// TwinCAT 3 PLC project Untitled1
// ProgramVersion: 3.1.4023.0
// libraries:
//   Tc2_Standard, * (Beckhoff Automation GmbH)
//   Tc2_System, * (Beckhoff Automation GmbH)
//   Tc2_Utilities, * (Beckhoff Automation GmbH)
//   Tc3_Module, * (Beckhoff Automation GmbH)
// project tree:
//   DUTs/ HMI_Button.TcDUT, HMI_Instructions.TcDUT, IO_Struct.TcDUT, Port_Map.TcDUT, SL_INSTRUCTIONS.TcDUT, Test_Log.TcDUT
//   GVLs/ GVL_HMI.TcGVL, GVL_IO_STRUCTS.TcGVL, GVL_LOGS.TcGVL, GVL_IO.TcGVL, CONSTANTS.TcGVL
//   / PlcTask.TcTTO
//   POUs/ FB_EXECUTE_SECTION1.TcPOU, FB_EXECUTE_SECTION2.TcPOU, INITIALIZE.TcPOU, LOG_SECTION2.TcPOU, LOG_SECTION1.TcPOU, MAIN.TcPOU, UNINITIALIZE.TcPOU, WRITE_IO_VALUES.TcPOU
// real-time tasks:
//   TASK PlcTask: cycle T#10ms, priority 20, ADS port 350
// I/O:
//   DEVICE Device 1 (EtherCAT), AmsNetId 169.254.202.152.2.1
//     C0 (EK1914) [EK1914, 2 Ch. Safety Input/Output 24V,  TwinSAFE]
//       modules: Module 1 (FSOE), Module 2 (DIO)
//       C1 (EL9410) [EL9410 E-Bus Power Supplier  (Diagnostics)]
//       C2 (EL2014) [EL2014 4Ch. Dig. Output 24V, 0,5A, Diagnostic]
//       C3 (EL1018) [EL1018 8Ch. Dig. Input 24V, 10µs]
//       C4 (EL1819) [EL1819 16Ch. Dig. Input 24V, 10µs]
//       C5 (EL1819) [EL1819 16Ch. Dig. Input 24V, 10µs]
//       C6 (EK1122-0008) [EK1122-0008 2 port EtherCAT junction M8]
//         JBC0 (EK1914) [EK1914, 2 Ch. Safety Input/Output 24V,  TwinSAFE]
//           modules: Module 1 (FSOE), Module 2 (DIO)
//           JBC1 (EL9410) [EL9410 E-Bus Power Supplier  (Diagnostics)]
//           JBC2 (EL1904) [EL1904, 4 Ch. Safety Input 24V, TwinSAFE]
//             modules: Module 1 (FSOES)
//           JBC3 (EL3174) [EL3174 4K. Ana. Eingang  +/-10V Diff., +/-20mA SingleEnded, 16 Bit]
//           JBC4 (EK1122-0008) [EK1122-0008 2 port EtherCAT junction M8]
//           JBC5 (EK1122-0008) [EK1122-0008 2 port EtherCAT junction M8]
//             Box 14 (EP3752-0000) [EP3752-0000 Acceleration Sensor]
// variable links:
//   Untitled1/Untitled1 Instance <-> Device 1 (EtherCAT)/C0 (EK1914)/C2 (EL2014)
//     PlcTask Outputs/GVL_IO.SF5_Fire_Alarm <-> DIG Outputs/Channel 2/Output
//   Untitled1/Untitled1 Instance <-> Device 1 (EtherCAT)/C0 (EK1914)/C3 (EL1018)
//     PlcTask Inputs/GVL_IO.J7_24V_Up <-> Channel 1/Input
//     PlcTask Inputs/GVL_IO.J8_24V_Up <-> Channel 3/Input
//     PlcTask Inputs/GVL_IO.J7_24V_Us <-> Channel 6/Input
//     PlcTask Inputs/GVL_IO.J8_24V_Us <-> Channel 8/Input
//   Untitled1/Untitled1 Instance <-> Device 1 (EtherCAT)/C0 (EK1914)/C4 (EL1819)
//     PlcTask Inputs/GVL_IO.J{1..6}_24V_Up <-> Channel {1..11 step 2}/Input  (6 links)
//     PlcTask Inputs/GVL_IO.J{1..6}_24V_Us <-> Channel {2..12 step 2}/Input  (6 links)
//   Untitled1/Untitled1 Instance <-> Device 1 (EtherCAT)/C0 (EK1914)/C5 (EL1819)
//     PlcTask Inputs/GVL_IO.SF1_MF_CONTINUITY <-> Channel 16/Input
//     PlcTask Inputs/GVL_IO.SF2_MF_CONTINUITY <-> Channel 15/Input
//     PlcTask Inputs/GVL_IO.SF4_Pull_Station <-> Channel 14/Input
//     PlcTask Inputs/GVL_IO.SF6_MGT_CONTINUITY <-> Channel 13/Input
//     PlcTask Inputs/GVL_IO.SF8_MGT_CONTINUITY <-> Channel 12/Input
//   Untitled1/Untitled1 Instance <-> Device 1 (EtherCAT)/C0 (EK1914)/C6 (EK1122-0008)/JBC0 (EK1914)
//     PlcTask Inputs/GVL_IO.JB_DCDCS_OK <-> Module 2 (DIO)/DIO Inputs/Input 0
//     PlcTask Inputs/GVL_IO.JB_Door_Switch <-> Module 2 (DIO)/DIO Inputs/Input 1
//     PlcTask Inputs/GVL_IO.JB_PSU1_OK <-> Module 2 (DIO)/DIO Inputs/Input 2
//     PlcTask Inputs/GVL_IO.JB_PSU2_OK <-> Module 2 (DIO)/DIO Inputs/Input 3

CONFIGURATION Untitled1
    RESOURCE PLC ON TwinCAT3
        TASK PlcTask(INTERVAL := T#10ms, PRIORITY := 20);
        PROGRAM MAIN WITH PlcTask : MAIN;
    END_RESOURCE
END_CONFIGURATION

// ---- DUTs/HMI_Button.TcDUT
TYPE HMI_Button :
STRUCT
	Text : STRING(50);
	Live_Value : BOOL;
END_STRUCT
END_TYPE

// ---- DUTs/HMI_Instructions.TcDUT
TYPE HMI_Instructions :
STRUCT
	Instructions : STRING(200);
	Status : BOOL;
END_STRUCT
END_TYPE

// ---- DUTs/IO_Struct.TcDUT
TYPE IO_Struct :
STRUCT
	SECTION : INT;
	INDEX : INT;
	CARD : STRING(10);
	TERMINAL : USINT;
	SCH_LBL : STRING(10);
	Signal : STRING(25);
	TESTER_PORT : STRING(10);
	TARGET_PORT : STRING(10);
	DESCRIPTION : STRING(255);
	LIVE_BOOL : BOOL;
	LIVE_INT : INT;
	EXPECTED_BOOL : BOOL;
	EXPECTED_INT : INT;
	RESULT : STRING(10);
END_STRUCT
END_TYPE

// ---- DUTs/Port_Map.TcDUT
TYPE Port_Map :
STRUCT
	JBOX_PORT : STRING(5);
	TESTER_PORT : STRING(5);
END_STRUCT
END_TYPE

// ---- DUTs/SL_INSTRUCTIONS.TcDUT
TYPE SL_INSTRUCTIONS :
STRUCT
	Line : STRING(255);
END_STRUCT
END_TYPE

// ---- DUTs/Test_Log.TcDUT
TYPE Test_Log :
STRUCT
	Index : INT;
	Description : STRING(255);
	Result : STRING(10);
END_STRUCT
END_TYPE

// ---- GVLs/GVL_HMI.TcGVL
{attribute 'qualified_only'}
VAR_GLOBAL
	
	JBOX_TEST_PORT_MAP : ARRAY[0..CONSTANTS.NUM_CONNECTIONS-1] OF Port_Map := [
		(
			JBOX_PORT := 'J37',
			TESTER_PORT := 'SF1'
		),
		(
			JBOX_PORT := 'S2',
			TESTER_PORT := 'SF2'
		),
		(
			JBOX_PORT := 'S33',
			TESTER_PORT := 'J1'
		),
		(
			JBOX_PORT := 'S34',
			TESTER_PORT := 'J2'
		),
		(
			JBOX_PORT := 'S25',
			TESTER_PORT := 'J3'
		),
		(
			JBOX_PORT := 'S26',
			TESTER_PORT := 'J4'
		),
		(
			JBOX_PORT := 'S27',
			TESTER_PORT := 'J5'
		),
		(
			JBOX_PORT := 'S28',
			TESTER_PORT := 'J6'
		),
		(
			JBOX_PORT := 'S29',
			TESTER_PORT := 'J7'
		),
		(
			JBOX_PORT := 'S30',
			TESTER_PORT := 'J8'
		),
		(
			JBOX_PORT := 'S1',
			TESTER_PORT := 'J9'
		),
		(*
		(
			JBOX_PORT := 'S35',
			TESTER_PORT := 'J10'
		),
		*)
		(
			JBOX_PORT := 'S3',
			TESTER_PORT := 'J11'
		),
		(
			JBOX_PORT := 'S5',
			TESTER_PORT := 'J12'
		),
		(
			JBOX_PORT := 'S8',
			TESTER_PORT := 'J13'
		),
		(
			JBOX_PORT := 'S10',
			TESTER_PORT := 'J14'
		),
		(
			JBOX_PORT := 'S21',
			TESTER_PORT := 'J15'
		),
		(
			JBOX_PORT := 'S22',
			TESTER_PORT := 'J16'
		),
		(
			JBOX_PORT := 'S23',
			TESTER_PORT := 'J17'
		),
		(
			JBOX_PORT := 'S24',
			TESTER_PORT := 'J18'
		),
		(
			JBOX_PORT := 'S4',
			TESTER_PORT := 'J19'
		),
		(
			JBOX_PORT := 'S6',
			TESTER_PORT := 'J20'
		),
		(
			JBOX_PORT := 'S9',
			TESTER_PORT := 'J21'
		),
		(
			JBOX_PORT := 'S11',
			TESTER_PORT := 'J22'
		),
		(
			JBOX_PORT := 'S13',
			TESTER_PORT := 'J23'
		),
		(
			JBOX_PORT := 'S14',
			TESTER_PORT := 'J24'
		),
		(
			JBOX_PORT := 'S15',
			TESTER_PORT := 'J25'
		),
		(
			JBOX_PORT := 'S16',
			TESTER_PORT := 'J26'
		),
		(
			JBOX_PORT := 'J36',
			TESTER_PORT := 'S17'
		)
		(*
		(
			JBOX_PORT := 'J38',
			TESTER_PORT := 'S18'
		)
		*)
		];

	//
	//
	//
	
	(*
	HMI_HOME_INSTRUCTIONS : ARRAY[0..1] OF HMI_INSTRUCTIONS := [
	];
	*)
	
	HMI_HOME_INSTRUCTIONS : ARRAY[0..CONSTANTS.HMI_HOME_NUM_INSTRUCTIONS-1] OF HMI_INSTRUCTIONS := [
		(Instructions := 'Place JBOX Next to Acceptance Tester',
		 Status := FALSE),
		(Instructions := 'Visually inspect the box for foreign objects, floating wires, or any signs of being incomplete',
		 Status := FALSE),
		(Instructions := 'Unplug power from the acceptance tester',
		 Status := FALSE),
		(Instructions := 'Verify green bonding wire is present to bond the door to the enclosure',
		 Status := FALSE),
		(Instructions := 'Connect All Tester Cables to JBOX Ports as Shown in the Port Map, Leave 120V Disconnected',
		 Status := FALSE),
		(Instructions := 'Open All Breakers in Acceptance Tester Panel',
		 Status := FALSE),
		(Instructions := 'Supply 480V Weld Plug on Acceptance Tester with 480V Power',
		 Status := FALSE),
		(Instructions := 'Close All Breakers in Acceptance Tester Panel',
		 Status := FALSE)
		 
	];
	
	HMI_HOME_BEGIN_TEST_BUTTON : HMI_BUTTON := (
		Text := 'Initiate JBOX Test',
		Live_Value := FALSE
	);
	
	HMI_SECTION_1_INSTRUCTIONS : ARRAY[0..CONSTANTS.HMI_SECTION_1_NUM_INSTRUCTIONS-1] OF HMI_INSTRUCTIONS := [
		(Instructions := 'Verify 480V Indicator for JBOX on Acceptance Tester',
		 Status := FALSE),
		(Instructions := 'Perform PSU1 Configuration',
		 Status := FALSE),
		(Instructions := 'Perform DCDC1 Configuration',
		 Status := FALSE),
		(Instructions := 'Perform DCDC2 Configuration',
		 Status := FALSE),
		(Instructions := 'Open JBOX Door',
		 Status := FALSE),
		(Instructions := 'Press Estop',
		 Status := FALSE),
		(Instructions := 'Pull Fire Alarm',
		 Status := FALSE)
	];
	
	HMI_PSU_CONFIG_INSTRUCTIONS : ARRAY[0..13] OF SL_INSTRUCTIONS := [
		(Line := 'Open the Phoenix Contact "Quint Power" App'),
		(Line := 'Install temportary 22 AWG jumper wire from PSU2 Rem signal to 0V TB'),
		(Line := 'Select READ VIA NFC'),
		(Line := 'Select SCAN VIA NFC'),
		(Line := 'Place top edge of phone over the QR code on PSU2 until power supply is read successfully'),
		(Line := 'Select OUTPUT VOLTAGE menu'),
		(Line := 'Set OUTPUT VOLTAGE to 26.00V'),
		(Line := 'Set PARALLEL OPERATION to TRUE'),
		(Line := 'Exit OUTPUT VOLTAGE menu and select SIGNALING menu'),
		(Line := 'Set OUT 2 to ANALOG OUTPUT with OUTPUT CURRENT'),
		(Line := 'Exit SIGNALING menu'),
		(Line := 'Select NFC button and plade top edge of phone over the QR code on PSU1 until the dara is written succesfully'),
		(Line := 'Remove temportary 22 AWG jumper wire FROM PSU2 Rem signal TO 0V TB'),
		(Line := 'Close Quint Power App')
	];
	
	HMI_DCDC_CONFIG_INSTRUCTIONS : ARRAY[0..3] OF SL_INSTRUCTIONS := [
		(Line := 'Pull ferrules inserted into terminals 2.1 and 2.2 in DC/DC slightly out so you can probe voltage on exposed ferrule'),
		(Line := 'Turn Uout dial on DC/DC2 until the DC/DCs output is 52V. Probe on exposed ferrules to verify'),
		(Line := 'Reseat ferrules to correct depth'),
		(Line := 'Write "52V, todays DATE, your initials" on the label on DC/DC')
	];

	
	
	HMI_SECTION_1_BEGIN_AUTOMATED_BUTTON : HMI_BUTTON := (
		Text := 'Begin Automated Test',
		Live_Value := FALSE
	);
	
	HMI_SECTION_2_INSTRUCTIONS : ARRAY[0..CONSTANTS.HMI_SECTION_2_NUM_INSTRUCTIONS-1] OF HMI_INSTRUCTIONS := [
		(Instructions := 'Reset Estop',
		 Status := FALSE),
		(Instructions := 'Reset Fire Alarm, use the key tied to the top of the acceptance tester to open the box and reset it',
		 Status := FALSE),
		(Instructions := 'Unplug J36 and S1 Connections on JBOX',
		 Status := FALSE),
		(Instructions := 'Plug J10 and S18 From Acceptance Tester into JBOX S35 and J38 Respectively',
		 Status := FALSE),
		(Instructions := 'Perform PSU2 Configuration',
		 Status := FALSE),
		(Instructions := 'Verify 120V Indicator for JBOX on Acceptance Tester',
		 Status := FALSE),
		(Instructions := 'Verify 120V Indicator FOR GRACE Port Verification Lit Up',
		 Status := FALSE),
		 (Instructions := 'Close JBOX Door',
		 Status := FALSE)
	];
	
	HMI_SECTION_2_BEGIN_AUTOMATED_BUTTON : HMI_BUTTON := (
		Text := 'Begin Automated Test',
		Live_Value := FALSE
	);
	
	
	HMI_ABORT_TEST_BUTTON : HMI_BUTTON := (
		Text := 'ABORT JBOX TEST',
		Live_Value := FALSE
	);
	
	HMI_RESET_TEST_BUTTON : HMI_BUTTON := (
		Text := 'Reset Jbox Test',
		Live_Value := FALSE
	);
	

	ACTIVE_HMI_VIEW_STRING : STRING(50);
	
	ACTIVE_HMI_VIEW : INT := 0;

	
	



	
	
END_VAR

// ---- GVLs/GVL_IO_STRUCTS.TcGVL
{attribute 'qualified_only'}
VAR_GLOBAL
	
	
	// STILL NEED ESTOP VERIFICATION, PSU VERIFICATION, DCDC VERIFICATION

	// SECTION ONE OCCURS WITH DOOR CLOSED AND ESTOP DEPRESSED AND NOTHING CONFIGURED
	IO_MAP_SECTION1_DIG : ARRAY[0..CONSTANTS.SECTION1_NUM_DIG_TESTS-1] OF IO_STRUCT := [
		(
			SECTION := 1,
			INDEX := 0,
			SCH_LBL := 'J7_4',
			SIGNAL := 'Digital',
			TESTER_PORT := 'J7',
			DESCRIPTION := '480V Supplied 7/8 S29 Up 24V Power Check', // This is written to HMI
			LIVE_BOOL := 0, // This is written to from the IO variable
			EXPECTED_BOOL := 1,
			RESULT := 'FAIL' // This is written from HMI
		),
		(
			SECTION := 1,
			INDEX := 1,
			SCH_LBL := 'J7_5',
			SIGNAL := 'Digital',
			TESTER_PORT := 'J7',
			DESCRIPTION := '480V Supplied 7/8 S29 Us 24V Power Check', // This is written to HMI
			LIVE_BOOL := 0, // This is written to from the IO variable
			EXPECTED_BOOL := 1,
			RESULT := 'FAIL' // This is written from HMI
		),
		(
			SECTION := 1,
			INDEX := 2,
			SCH_LBL := 'J8_4',
			SIGNAL := 'Digital',
			TESTER_PORT := 'J8',
			DESCRIPTION := '480V Supplied 7/8 S30 Up 24V Power Check', // This is written to HMI
			LIVE_BOOL := 0, // This is written to from the IO variable
			EXPECTED_BOOL := 1,
			RESULT := 'FAIL' // This is written from HMI
		),
		(
			SECTION := 1,
			INDEX := 3,
			SCH_LBL := 'J8_5',
			SIGNAL := 'Digital',
			TESTER_PORT := 'J8',
			DESCRIPTION := '480V Supplied 7/8 S30 Us 24V Power Check', // This is written to HMI
			LIVE_BOOL := 0, // This is written to from the IO variable
			EXPECTED_BOOL := 1,
			RESULT := 'FAIL' // This is written from HMI
		),
		(
			SECTION := 1,
			INDEX := 4,
			SCH_LBL := 'J1_1',
			SIGNAL := 'Digital',
			TESTER_PORT := 'J1',
			DESCRIPTION := '480V Supplied 24V Lighting Up S33', // This is written to HMI
			LIVE_BOOL := 0, // This is written to from the IO variable
			EXPECTED_BOOL := 1,
			RESULT := 'FAIL' // This is written from HMI
		),
		(
			SECTION := 1,
			INDEX := 5,
			SCH_LBL := 'J1_2',
			SIGNAL := 'Digital',
			TESTER_PORT := 'J1',
			DESCRIPTION := '480V Supplied 24V Lighting Up S33', // This is written to HMI
			LIVE_BOOL := 0, // This is written to from the IO variable
			EXPECTED_BOOL := 1,
			RESULT := 'FAIL' // This is written from HMI
		),
		(
			SECTION := 1,
			INDEX := 6,
			SCH_LBL := 'J2_1',
			SIGNAL := 'Digital',
			TESTER_PORT := 'J2',
			DESCRIPTION := '480V Supplied 24V Lighting Up S34', // This is written to HMI
			LIVE_BOOL := 0, // This is written to from the IO variable
			EXPECTED_BOOL := 1,
			RESULT := 'FAIL' // This is written from HMI
		),
		(
			SECTION := 1,
			INDEX := 7,
			SCH_LBL := 'J2_2',
			SIGNAL := 'Digital',
			TESTER_PORT := 'J2',
			DESCRIPTION := '480V Supplied 24V Lighting Us S34', // This is written to HMI
			LIVE_BOOL := 0, // This is written to from the IO variable
			EXPECTED_BOOL := 1,
			RESULT := 'FAIL' // This is written from HMI
		),
		(
			SECTION := 1,
			INDEX := 8,
			SCH_LBL := 'J3_1',
			SIGNAL := 'Digital',
			TESTER_PORT := 'J3',
			DESCRIPTION := '480V Supplied 24V Lighting Up S25', // This is written to HMI
			LIVE_BOOL := 0, // This is written to from the IO variable
			EXPECTED_BOOL := 1,
			RESULT := 'FAIL' // This is written from HMI
		),
		(
			SECTION := 1,
			INDEX := 9,
			SCH_LBL := 'J3_2',
			SIGNAL := 'Digital',
			TESTER_PORT := 'J3',
			DESCRIPTION := '480V Supplied 24V Lighting Us S25', // This is written to HMI
			LIVE_BOOL := 0, // This is written to from the IO variable
			EXPECTED_BOOL := 1,
			RESULT := 'FAIL' // This is written from HMI
		),
		(
			SECTION := 1,
			INDEX := 10,
			SCH_LBL := 'J4_1',
			SIGNAL := 'Digital',
			TESTER_PORT := 'J4',
			DESCRIPTION := '480V Supplied 24V Lighting Up S26', // This is written to HMI
			LIVE_BOOL := 0, // This is written to from the IO variable
			EXPECTED_BOOL := 1,
			RESULT := 'FAIL' // This is written from HMI
		),
		(
			SECTION := 1,
			INDEX := 11,
			SCH_LBL := 'J4_2',
			SIGNAL := 'Digital',
			TESTER_PORT := 'J4',
			DESCRIPTION := '480V Supplied 24V Lighting Us S26', // This is written to HMI
			LIVE_BOOL := 0, // This is written to from the IO variable
			EXPECTED_BOOL := 1,
			RESULT := 'FAIL' // This is written from HMI
		),
		(
			SECTION := 1,
			INDEX := 12,
			SCH_LBL := 'J5_1',
			SIGNAL := 'Digital',
			TESTER_PORT := 'J5',
			DESCRIPTION := '480V Supplied 24V Lighting Up S27', // This is written to HMI
			LIVE_BOOL := 0, // This is written to from the IO variable
			EXPECTED_BOOL := 1,
			RESULT := 'FAIL' // This is written from HMI
		),
		(
			SECTION := 1,
			INDEX := 13,
			SCH_LBL := 'J5_2',
			SIGNAL := 'Digital',
			TESTER_PORT := 'J5',
			DESCRIPTION := '480V Supplied 24V Lighting Us S27', // This is written to HMI
			LIVE_BOOL := 0, // This is written to from the IO variable
			EXPECTED_BOOL := 1,
			RESULT := 'FAIL' // This is written from HMI
		),
		(
			SECTION := 1,
			INDEX := 14,
			SCH_LBL := 'J6_1',
			SIGNAL := 'Digital',
			TESTER_PORT := 'J6',
			DESCRIPTION := '480V Supplied 24V Lighting Up S28', // This is written to HMI
			LIVE_BOOL := 0, // This is written to from the IO variable
			EXPECTED_BOOL := 1,
			RESULT := 'FAIL' // This is written from HMI
		),
		(
			SECTION := 1,
			INDEX := 15,
			SCH_LBL := 'J6_2',
			SIGNAL := 'Digital',
			TESTER_PORT := 'J6',
			DESCRIPTION := '480V Supplied 24V Lighting Us S28', // This is written to HMI
			LIVE_BOOL := 0, // This is written to from the IO variable
			EXPECTED_BOOL := 1,
			RESULT := 'FAIL' // This is written from HMI
		),
		(
			SECTION := 1,
			INDEX := 16,
			SCH_LBL := 'SF1',
			SIGNAL := 'Digital',
			TESTER_PORT := 'SF2',
			TARGET_PORT := 'S2',
			DESCRIPTION := 'Mine Phone Continuity SF1', // This is written to HMI
			LIVE_BOOL := 0, // This is written to from the IO variable
			EXPECTED_BOOL := 1,
			RESULT := 'FAIL' // This is written from HMI
		),
		(
			SECTION := 1,
			INDEX := 17,
			SCH_LBL := 'SF2',
			SIGNAL := 'Digital',
			TESTER_PORT := 'SF2',
			TARGET_PORT := 'S2',
			DESCRIPTION := 'Mine Phone Continuity SF2', // This is written to HMI
			LIVE_BOOL := 0, // This is written to from the IO variable
			EXPECTED_BOOL := 1,
			RESULT := 'FAIL' // This is written from HMI
		),
		(
			SECTION := 1,
			INDEX := 18,
			SCH_LBL := 'SF4',
			SIGNAL := 'Digital',
			TESTER_PORT := 'SF2',
			TARGET_PORT := 'S2',
			DESCRIPTION := 'Fire Pull Station Pulled', // This is written to HMI
			LIVE_BOOL := 0, // This is written to from the IO variable
			EXPECTED_BOOL := 0,
			RESULT := 'FAIL' // This is written from HMI
		),
		(
			SECTION := 1,
			INDEX := 19,
			SCH_LBL := 'SF6',
			SIGNAL := 'Digital',
			TESTER_PORT := 'SF2',
			TARGET_PORT := 'S2',
			DESCRIPTION := 'MGT Continuity SF6', // This is written to HMI
			LIVE_BOOL := 0, // This is written to from the IO variable
			EXPECTED_BOOL := 1,
			RESULT := 'FAIL' // This is written from HMI
		),
		(
			SECTION := 1,
			INDEX := 20,
			SCH_LBL := 'SF8',
			SIGNAL := 'Digital',
			TESTER_PORT := 'SF2',
			TARGET_PORT := 'S2',
			DESCRIPTION := 'MGT Continuity SF8', // This is written to HMI
			LIVE_BOOL := 0, // This is written to from the IO variable
			EXPECTED_BOOL := 1,
			RESULT := 'FAIL' // This is written from HMI
		),
		(
			SECTION := 1,
			INDEX := 21,
			SIGNAL := 'Digital',
			DESCRIPTION := 'JBOX Door Switch Open', // This is written to HMI
			LIVE_BOOL := 0, // This is written to from the IO variable
			EXPECTED_BOOL := 0,
			RESULT := 'FAIL' // This is written from HMI
		),
		(
			SECTION := 1,
			INDEX := 22,
			SIGNAL := 'Digital',
			DESCRIPTION := 'JBOX DCDCs_OK', // This is written to HMI
			LIVE_BOOL := 0, // This is written to from the IO variable
			EXPECTED_BOOL := 1,
			RESULT := 'FAIL' // This is written from HMI
		),
		(
			SECTION := 1,
			INDEX := 23,
			SIGNAL := 'Digital',
			DESCRIPTION := 'JBOX PSU2_OK', // This is written to HMI
			LIVE_BOOL := 0, // This is written to from the IO variable
			EXPECTED_BOOL := 1,
			RESULT := 'FAIL' // This is written from HMI
		)
		
	];
	
	IO_MAP_SECTION1_HMI : ARRAY[0..CONSTANTS.SECTION1_NUM_HMI_TESTS-1] OF IO_STRUCT := [
		(
			SECTION := 1,
			SIGNAL := 'HMI',
			TESTER_PORT := 'J2',
			DESCRIPTION := 'JBOX 480V Test', // This is written to HMI
			LIVE_BOOL := 0, // This is written to from the IO variable
			EXPECTED_BOOL := 1,
			RESULT := 'FAIL' // This is written from HMI
		),
		(
			SECTION := 1,
			DESCRIPTION := 'Performed PSU1 Configuration', // This is written to HMI
			LIVE_BOOL := 0, // This is written to from the IO variable
			EXPECTED_BOOL := 1,
			RESULT := 'FAIL' // This is written from HMI
		),
		(
			SECTION := 1,
			DESCRIPTION := 'Performed DCDC1 Configuration', // This is written to HMI
			LIVE_BOOL := 0, // This is written to from the IO variable
			EXPECTED_BOOL := 1,
			RESULT := 'FAIL' // This is written from HMI
		),
		(
			SECTION := 1,
			DESCRIPTION := 'Performed DCDC2 Configuration', // This is written to HMI
			LIVE_BOOL := 0, // This is written to from the IO variable
			EXPECTED_BOOL := 1,
			RESULT := 'FAIL' // This is written from HMI
		)
		
		(*
		(
			SECTION := 1,
			INDEX := 1,
			CARD := '',
			// TERMINAL := NULL,
			SCH_LBL := '',
			SIGNAL := 'HMI',
			TESTER_PORT := '',
			TARGET_PORT := '',
			DESCRIPTION := 'JBOX 120V Test', // This is written to HMI
			LIVE_BOOL := 0, // This is written to from the IO variable
			EXPECTED_BOOL := 1,
			RESULT := 'FAIL' // This is written from HMI
		)
		*)
	];
	

	// SECTION TWO OCCURS WITH DOOR OPEN, ESTOP PRESSED, AND PULL STATION PULLED
	// Need to get Estop Stuff In Here
	IO_MAP_SECTION2_DIG : ARRAY[0..CONSTANTS.SECTION2_NUM_DIG_TESTS-1] OF IO_STRUCT := [
		(
			SECTION := 2,
			INDEX := 0,
			CARD := 'C3',
			TERMINAL :=  1,
			SCH_LBL := 'SF4',
			SIGNAL := 'Digital',
			TESTER_PORT := 'SF2',
			TARGET_PORT := 'S2',
			DESCRIPTION := 'Fire Pull Station Reset Verification', // This is written to HMI
			LIVE_BOOL := 0, // This is written to from the IO variable
			EXPECTED_BOOL := 1,
			RESULT := 'FAIL' // This is written from HMI
		),
		(
			SECTION := 2,
			INDEX := 1,
			CARD := 'JBC0',
			TERMINAL :=  10,
			SCH_LBL := '',
			SIGNAL := 'Digital',
			TESTER_PORT := '',
			TARGET_PORT := '',
			DESCRIPTION := 'Door Switch Closed Verification', // This is written to HMI
			LIVE_BOOL := 0, // This is written to from the IO variable
			EXPECTED_BOOL := 1,
			RESULT := 'FAIL' // This is written from HMI
		),
		(
			SECTION := 1,
			INDEX := 2,
			SIGNAL := 'Digital',
			DESCRIPTION := 'JBOX PSU1_OK', // This is written to HMI
			LIVE_BOOL := 0, // This is written to from the IO variable
			EXPECTED_BOOL := 1,
			RESULT := 'FAIL' // This is written from HMI
		),
		(
			SECTION := 1,
			INDEX := 3,
			SCH_LBL := 'J7_4',
			SIGNAL := 'Digital',
			TESTER_PORT := 'J7',
			DESCRIPTION := '120V Supplied 7/8 S29 Up 24V Power Check', // This is written to HMI
			LIVE_BOOL := 0, // This is written to from the IO variable
			EXPECTED_BOOL := 1,
			RESULT := 'FAIL' // This is written from HMI
		),
		(
			SECTION := 1,
			INDEX := 4,
			SCH_LBL := 'J7_5',
			SIGNAL := 'Digital',
			TESTER_PORT := 'J7',
			DESCRIPTION := '120V Supplied 7/8 S29 Us 24V Power Check', // This is written to HMI
			LIVE_BOOL := 0, // This is written to from the IO variable
			EXPECTED_BOOL := 1,
			RESULT := 'FAIL' // This is written from HMI
		),
		(
			SECTION := 1,
			INDEX := 5,
			SCH_LBL := 'J8_4',
			SIGNAL := 'Digital',
			TESTER_PORT := 'J8',
			DESCRIPTION := '120V Supplied 7/8 S30 Up 24V Power Check', // This is written to HMI
			LIVE_BOOL := 0, // This is written to from the IO variable
			EXPECTED_BOOL := 1,
			RESULT := 'FAIL' // This is written from HMI
		),
		(
			SECTION := 1,
			INDEX := 6,
			SCH_LBL := 'J8_5',
			SIGNAL := 'Digital',
			TESTER_PORT := 'J8',
			DESCRIPTION := '120V Supplied 7/8 S30 Us 24V Power Check', // This is written to HMI
			LIVE_BOOL := 0, // This is written to from the IO variable
			EXPECTED_BOOL := 1,
			RESULT := 'FAIL' // This is written from HMI
		),
		(
			SECTION := 1,
			INDEX := 7,
			SCH_LBL := 'J1_1',
			SIGNAL := 'Digital',
			TESTER_PORT := 'J1',
			DESCRIPTION := '120V Supplied 24V Lighting Up S33', // This is written to HMI
			LIVE_BOOL := 0, // This is written to from the IO variable
			EXPECTED_BOOL := 1,
			RESULT := 'FAIL' // This is written from HMI
		),
		(
			SECTION := 1,
			INDEX := 8,
			SCH_LBL := 'J1_2',
			SIGNAL := 'Digital',
			TESTER_PORT := 'J1',
			DESCRIPTION := '120V Supplied 24V Lighting Up S33', // This is written to HMI
			LIVE_BOOL := 0, // This is written to from the IO variable
			EXPECTED_BOOL := 1,
			RESULT := 'FAIL' // This is written from HMI
		),
		(
			SECTION := 1,
			INDEX := 9,
			SCH_LBL := 'J2_1',
			SIGNAL := 'Digital',
			TESTER_PORT := 'J2',
			DESCRIPTION := '120V Supplied 24V Lighting Up S34', // This is written to HMI
			LIVE_BOOL := 0, // This is written to from the IO variable
			EXPECTED_BOOL := 1,
			RESULT := 'FAIL' // This is written from HMI
		),
		(
			SECTION := 1,
			INDEX := 10,
			SCH_LBL := 'J2_2',
			SIGNAL := 'Digital',
			TESTER_PORT := 'J2',
			DESCRIPTION := '120V Supplied 24V Lighting Us S34', // This is written to HMI
			LIVE_BOOL := 0, // This is written to from the IO variable
			EXPECTED_BOOL := 1,
			RESULT := 'FAIL' // This is written from HMI
		),
		(
			SECTION := 1,
			INDEX := 11,
			SCH_LBL := 'J3_1',
			SIGNAL := 'Digital',
			TESTER_PORT := 'J3',
			DESCRIPTION := '120V Supplied 24V Lighting Up S25', // This is written to HMI
			LIVE_BOOL := 0, // This is written to from the IO variable
			EXPECTED_BOOL := 1,
			RESULT := 'FAIL' // This is written from HMI
		),
		(
			SECTION := 1,
			INDEX := 12,
			SCH_LBL := 'J3_2',
			SIGNAL := 'Digital',
			TESTER_PORT := 'J3',
			DESCRIPTION := '120V Supplied 24V Lighting Us S25', // This is written to HMI
			LIVE_BOOL := 0, // This is written to from the IO variable
			EXPECTED_BOOL := 1,
			RESULT := 'FAIL' // This is written from HMI
		),
		(
			SECTION := 1,
			INDEX := 13,
			SCH_LBL := 'J4_1',
			SIGNAL := 'Digital',
			TESTER_PORT := 'J4',
			DESCRIPTION := '120V Supplied 24V Lighting Up S26', // This is written to HMI
			LIVE_BOOL := 0, // This is written to from the IO variable
			EXPECTED_BOOL := 1,
			RESULT := 'FAIL' // This is written from HMI
		),
		(
			SECTION := 1,
			INDEX := 14,
			SCH_LBL := 'J4_2',
			SIGNAL := 'Digital',
			TESTER_PORT := 'J4',
			DESCRIPTION := '120V Supplied 24V Lighting Us S26', // This is written to HMI
			LIVE_BOOL := 0, // This is written to from the IO variable
			EXPECTED_BOOL := 1,
			RESULT := 'FAIL' // This is written from HMI
		),
		(
			SECTION := 1,
			INDEX := 15,
			SCH_LBL := 'J5_1',
			SIGNAL := 'Digital',
			TESTER_PORT := 'J5',
			DESCRIPTION := '120V Supplied 24V Lighting Up S27', // This is written to HMI
			LIVE_BOOL := 0, // This is written to from the IO variable
			EXPECTED_BOOL := 1,
			RESULT := 'FAIL' // This is written from HMI
		),
		(
			SECTION := 1,
			INDEX := 16,
			SCH_LBL := 'J5_2',
			SIGNAL := 'Digital',
			TESTER_PORT := 'J5',
			DESCRIPTION := '120V Supplied 24V Lighting Us S27', // This is written to HMI
			LIVE_BOOL := 0, // This is written to from the IO variable
			EXPECTED_BOOL := 1,
			RESULT := 'FAIL' // This is written from HMI
		),
		(
			SECTION := 1,
			INDEX := 17,
			SCH_LBL := 'J6_1',
			SIGNAL := 'Digital',
			TESTER_PORT := 'J6',
			DESCRIPTION := '120V Supplied 24V Lighting Up S28', // This is written to HMI
			LIVE_BOOL := 0, // This is written to from the IO variable
			EXPECTED_BOOL := 1,
			RESULT := 'FAIL' // This is written from HMI
		),
		(
			SECTION := 1,
			INDEX := 18,
			SCH_LBL := 'J6_2',
			SIGNAL := 'Digital',
			TESTER_PORT := 'J6',
			DESCRIPTION := '120V Supplied 24V Lighting Us S28', // This is written to HMI
			LIVE_BOOL := 0, // This is written to from the IO variable
			EXPECTED_BOOL := 1,
			RESULT := 'FAIL' // This is written from HMI
		)
		];
		
	

	IO_MAP_SECTION2_HMI : ARRAY[0..CONSTANTS.SECTION2_NUM_HMI_TESTS-1] OF IO_STRUCT := [
		(
			SECTION := 1,
			INDEX := 0,
			SIGNAL := 'HMI',
			DESCRIPTION := 'Performed PSU2 Configuration', // This is written to HMI
			LIVE_BOOL := 0, // This is written to from the IO variable
			EXPECTED_BOOL := 1,
			RESULT := 'FAIL' // This is written from HMI
		),
		(
			SECTION := 1,
			INDEX := 1,
			SIGNAL := 'HMI',
			DESCRIPTION := '120V Grace Port Lit Up', // This is written to HMI
			LIVE_BOOL := 0, // This is written to from the IO variable
			EXPECTED_BOOL := 1,
			RESULT := 'FAIL' // This is written from HMI
		),
		(
			SECTION := 1,
			INDEX := 2,
			SIGNAL := 'HMI',
			DESCRIPTION := '120V Grace outlet verification grace lit up', // This is written to HMI
			LIVE_BOOL := 0, // This is written to from the IO variable
			EXPECTED_BOOL := 1,
			RESULT := 'FAIL' // This is written from HMI
		)
		];

END_VAR

// ---- GVLs/GVL_LOGS.TcGVL
{attribute 'qualified_only'}
VAR_GLOBAL
	// All JBOX Connectors are Plugged In, Door Closed, Estop Depressed, Fire Alarm Nominal
	TEST_RESULTS_ARRAY : ARRAY[0..CONSTANTS.TOTAL_NUM_TESTS-1] OF Test_Log; 
		
	NUM_TESTS_LOGGED : INT;
END_VAR

// ---- GVLs/GVL_IO.TcGVL
{attribute 'qualified_only'}
VAR_GLOBAL
	
	SECTION1_DIG_INPUTS : ARRAY[0..CONSTANTS.SECTION1_NUM_DIG_TESTS-1] OF POINTER TO BOOL;
	
	SECTION2_DIG_INPUTS : ARRAY[0..CONSTANTS.SECTION2_NUM_DIG_TESTS-1] OF POINTER TO BOOL;
	
	{attribute 'TcLinkTo' := 'TIIB[C3 (EL1018)]^Channel 1^Input'}
	J7_24V_Up AT%I* : BOOL; //14.1 : BOOL; (*INDEX 4 24V PWR Check J7 (4) (1008 (1) port 2) *)
    {attribute 'TcLinkTo' := 'TIIB[C3 (EL1018)]^Channel 6^Input'}
	J7_24V_Us AT%I* : BOOL; //4.2 : BOOL; (*INDEX 5 24V PWR Check J7 (5) (1008 (1) port 3) *)    
	{attribute 'TcLinkTo' := 'TIIB[C3 (EL1018)]^Channel 3^Input'}
	J8_24V_Up AT%I* : BOOL; //5.4 : BOOL; (*INDEX 14 24V PWR Check J8 (4) (1008 (2) port 5) *)
    {attribute 'TcLinkTo' := 'TIIB[C3 (EL1018)]^Channel 8^Input'}
	J8_24V_Us AT%I* : BOOL; //5.5 : BOOL; (*INDEX 15 24V PWR Check J8 (5) (1008 (2) port 6) *)

	
	
	{attribute 'TcLinkTo' := 'TIIB[C4 (EL1819)]^Channel 1^Input'}	
	J1_24V_Up AT%I* : BOOL; //6.2 : BOOL; (*INDEX 20 Lighting 24V Check J1 (1) (1008 (3) port 3) *)
	{attribute 'TcLinkTo' := 'TIIB[C4 (EL1819)]^Channel 2^Input'}	
	J1_24V_Us AT%I* : BOOL; //6.3 : BOOL; (*INDEX 21 Lighting 24V Check J1 (2) (1008 (3) port 4) *)
	{attribute 'TcLinkTo' := 'TIIB[C4 (EL1819)]^Channel 3^Input'}	
	J2_24V_Up AT%I* : BOOL; //6.4 : BOOL; (*INDEX 22 Lighting 24V Check J2 (1) (1008 (3) port 5) *)
	{attribute 'TcLinkTo' := 'TIIB[C4 (EL1819)]^Channel 4^Input'}	
	J2_24V_Us AT%I* : BOOL; //6.5 : BOOL; (*INDEX 23 Lighting 24V Check J2 (2) (1008 (3) port 6) *)
	{attribute 'TcLinkTo' := 'TIIB[C4 (EL1819)]^Channel 5^Input'}	
	J3_24V_Up AT%I* : BOOL; //14.3 : BOOL; (*INDEX 6 24V PWR Check J3 (1) (1008 (1) port 4) *)
	{attribute 'TcLinkTo' := 'TIIB[C4 (EL1819)]^Channel 6^Input'}	
	J3_24V_Us AT%I* : BOOL; //4.4 : BOOL; (*INDEX 7 24V PWR Check J3 (2) (1008 (1) port 5) *)
	{attribute 'TcLinkTo' := 'TIIB[C4 (EL1819)]^Channel 7^Input'}	
	J4_24V_Up AT%I* : BOOL; //4.5 : BOOL; (*INDEX 8 24V PWR Check J4 (1) (1008 (1) port 6) *)
	{attribute 'TcLinkTo' := 'TIIB[C4 (EL1819)]^Channel 8^Input'}	
    J4_24V_Us AT%I* : BOOL; //4.7 : BOOL; (*INDEX 9 24V PWR Check J4 (2) (1008 (1) port 7) *)
	{attribute 'TcLinkTo' := 'TIIB[C4 (EL1819)]^Channel 9^Input'}	
	J5_24V_Up AT%I* : BOOL; //5.0 : BOOL; (*INDEX 10 24V PWR Check J5 (1) (1008 (2) port 1) *)
	{attribute 'TcLinkTo' := 'TIIB[C4 (EL1819)]^Channel 10^Input'}	
	J5_24V_Us AT%I* : BOOL; //5.1 : BOOL; (*INDEX 11 24V PWR Check J5 (2) (1008 (2) port 2) *)
	{attribute 'TcLinkTo' := 'TIIB[C4 (EL1819)]^Channel 11^Input'}	
	J6_24V_Up AT%I* : BOOL; //5.2 : BOOL; (*INDEX 12 24V PWR Check J6 (1) (1008 (2) port 3) *)
	{attribute 'TcLinkTo' := 'TIIB[C4 (EL1819)]^Channel 12^Input'}	
	J6_24V_Us AT%I* : BOOL; //5.3 : BOOL; (*INDEX 13 24V PWR Check J6 (2) (1008 (2) port 4) *)
	
	
	{attribute 'TcLinkTo' := 'TIIB[C5 (EL1819)]^Channel 16^Input'}	
	SF1_MF_CONTINUITY AT%I* : BOOL; //5.7 : BOOL; (*INDEX 17 Mine Phone Continuity SF1 (1008 (2) port 8) *)
	{attribute 'TcLinkTo' := 'TIIB[C5 (EL1819)]^Channel 15^Input'}	
	SF2_MF_CONTINUITY AT%I* : BOOL; //5.6 : BOOL; (*INDEX 16 Mine Phone Continuity SF2 (1008 (2) port 7) *)	
	{attribute 'TcLinkTo' := 'TIIB[C5 (EL1819)]^Channel 14^Input'}	
	SF4_Pull_Station AT%I* : BOOL; //4.0 : BOOL; (*INDEX 3 Fire pull Station SF4 (1008 (1) port 1) *)	
	{attribute 'TcLinkTo' := 'TIIB[C5 (EL1819)]^Channel 13^Input'}	
	SF6_MGT_CONTINUITY AT%I* : BOOL; //6.0 : BOOL; (*INDEX 18 MGT Continuity SF6 (1008 (3) port 1) *)
	{attribute 'TcLinkTo' := 'TIIB[C5 (EL1819)]^Channel 12^Input'}	
	SF8_MGT_CONTINUITY AT%I* : BOOL; //6.1: BOOL; (*INDEX 19 MGT Continuity SF8 (1008 (3) port 2) *)

	{attribute 'TcLinkTo' := 'TIIB[JBC0 (EK1914)]^Module 2 (DIO)^DIO Inputs^Input 1'}
	JB_Door_Switch AT%I* : BOOL; (* Door Switch *)
	
	{attribute 'TcLinkTo' := 'TIIB[JBC0 (EK1914)]^Module 2 (DIO)^DIO Inputs^Input 0'}
	JB_DCDCS_OK AT%I* : BOOL; (* JBOX DCDC GOOD Signal *)
	
	{attribute 'TcLinkTo' := 'TIIB[JBC0 (EK1914)]^Module 2 (DIO)^DIO Inputs^Input 2'}
	JB_PSU1_OK AT%I* : BOOL; (* PSU 1 OK *)
	
	{attribute 'TcLinkTo' := 'TIIB[JBC0 (EK1914)]^Module 2 (DIO)^DIO Inputs^Input 3'}
	JB_PSU2_OK AT%I* : BOOL; (* PSU 2 OK *)
	
	
	{attribute 'TcLinkTo' := 'TIIB[C2 (EL2014)]^DIG Outputs^Channel 2^Output'}
	SF5_Fire_Alarm AT%Q* : BOOL; //3.1 : BOOL; (*INDEX 0 Fire Alarm Sound SF5 (2024 port 2) *)
	



	//JB_1914_Us AT%I* : BOOL; //8.0 : BOOL; (*INDEX 1 JBOX 1914 Up Power *) // mapping is likely wrong
	//JB_1914_Up AT%I* : BOOL; //8.1 : BOOL; (*INDEX 2 JBOX 1914 Us Power *) // mapping is likely wrong

	
	//PSU1_Stat AT%I* : BOOL; //8.2 : BOOL; (*INDEX 24 PSU1_OK/1.4B *)
	
	//PSU2_Stat AT%I* : BOOL; //8.3 : BOOL; (*INDEX 25 PSU2_OK/1.4E *)
	
    
	//PSU1_I AT%I* : BOOL; //10.0 : BOOL; (*INDEX 26 PSU1_IOUT/1.3B *)
    
	//PSU2_I AT%I* : BOOL; //10.1 : BOOL; (*INDEX 27 PSU2_IOUT/1.3E *)
	
	// MAYBE BADDD JBC0_P2 AT%I45.0 : BOOL; (* DCDC_OK/1.6C *)
    
	
	
	
	// INCLINOMETERRRRRR
	
	
	(* FIGURE OUT SAFETY STUFF
	

    JBC0_P7 AT%I40.0 : BOOL; (* SAFE_IN1_I *)
    JBC0_P15 AT%I* : BOOL; (* SAFE_IN2_I *)
    JBC0_P6 AT%I* : BOOL; (* SAFE_IN1_O *)
    JBC0_P14 AT%I* : BOOL; (* SAFE_IN2_O *)
    
   
	*)
	
	
	
	(* MAYBE TEST AND DO THIS FOR THE REST OF THE JBOX CARDS
	
	JB_2014_DIAG_1 AT%I61 : BOOL; (* PSU2_IOUT/1.3E *)
	JB_2014_DIAG_2 AT%I61.4 : BOOL; (* PSU2_IOUT/1.3E *)
	JB_2014_DIAG_3 AT%I62 : BOOL; (* PSU2_IOUT/1.3E *)
	JB_2014_DIAG_4 AT%I62.4 : BOOL; (* PSU2_IOUT/1.3E *)
	JB_2014_COM_FAULT AT%I63.0 : BOOL; (* PSU2_IOUT/1.3E *)
	JB_2014_OVERTEMP AT%I63.1 : BOOL; (* PSU2_IOUT/1.3E *)
	JB_2014_UNDERVOLT AT%I63.2 : BOOL; (* PSU2_IOUT/1.3E *)
	JB_2014_MISS_VOLT AT%I63.3 : BOOL; (* PSU2_IOUT/1.3E *)
	*)


END_VAR

// ---- GVLs/CONSTANTS.TcGVL
{attribute 'qualified_only'}
VAR_GLOBAL CONSTANT

	
	HMI_HOME_NUM_INSTRUCTIONS : INT := 8;
	
	HMI_SECTION_1_NUM_INSTRUCTIONS : INT := 7;
	
	HMI_SECTION_2_NUM_INSTRUCTIONS : INT := 8;
	
	TOTAL_NUM_TESTS : INT := 70;
	
	SECTION1_NUM_DIG_TESTS : INT := 24;
	
	SECTION1_NUM_HMI_TESTS : INT := 4;
	
	SECTION2_NUM_DIG_TESTS : INT := 19;
	
	SECTION2_NUM_HMI_TESTS : INT := 3;
	
	NUM_CONNECTIONS : INT := 28;
	
END_VAR

// ---- POUs/MAIN.TcPOU
PROGRAM MAIN
VAR_INPUT
END_VAR
VAR
	ExecuteSection1 : FB_EXECUTE_SECTION1;
	ExecuteSection2 : FB_EXECUTE_SECTION2;
	
	temp_ver_value : BOOL;

	i : INT;
	
	Delay : TON;
	Delay1 : TON;
	
	
END_VAR


IF GVL_HMI.HMI_ABORT_TEST_BUTTON.Live_Value THEN
	UNINITIALIZE();
END_IF

CASE GVL_HMI.ACTIVE_HMI_VIEW OF
  0: GVL_HMI.ACTIVE_HMI_VIEW_STRING := 'Home_Page.content';
  1: GVL_HMI.ACTIVE_HMI_VIEW_STRING := 'Section_1.content';
  2: GVL_HMI.ACTIVE_HMI_VIEW_STRING := 'Section_2.content';
  3: GVL_HMI.ACTIVE_HMI_VIEW_STRING := 'Results_Page.content';
  11: GVL_HMI.ACTIVE_HMI_VIEW_STRING := 'Section_1.content';
  12: GVL_HMI.ACTIVE_HMI_VIEW_STRING := 'Section_2.content';
  ELSE GVL_HMI.ACTIVE_HMI_VIEW_STRING := 'Home_Page.content';  // default
END_CASE;

CASE GVL_HMI.ACTIVE_HMI_VIEW OF
	
	0: // Idle
	
		Initialize();
		
		temp_ver_value := TRUE;
		
		FOR i := 0 TO CONSTANTS.HMI_HOME_NUM_INSTRUCTIONS - 1 DO
			IF GVL_HMI.HMI_HOME_INSTRUCTIONS[i].Status = FALSE THEN
				temp_ver_value := FALSE;
			END_IF
		END_FOR
		
		IF GVL_HMI.HMI_HOME_BEGIN_TEST_BUTTON.Live_Value AND temp_ver_value THEN
			GVL_HMI.ACTIVE_HMI_VIEW := 1;
		END_IF
		

	1: 
	
		temp_ver_value := TRUE;
		
		FOR i := 0 TO CONSTANTS.HMI_SECTION_1_NUM_INSTRUCTIONS - 1 DO
			IF GVL_HMI.HMI_SECTION_1_INSTRUCTIONS[i].Status = FALSE THEN
				temp_ver_value := FALSE;
			END_IF
		END_FOR
		
		IF GVL_HMI.HMI_SECTION_1_BEGIN_AUTOMATED_BUTTON.Live_Value AND temp_ver_value THEN
			GVL_HMI.ACTIVE_HMI_VIEW := 11;

		END_IF
		
	2:
	
		temp_ver_value := TRUE;
		
		FOR I:= 0 TO CONSTANTS.HMI_SECTION_2_NUM_INSTRUCTIONS - 1 DO
			IF GVL_HMI.HMI_SECTION_2_INSTRUCTIONS[i].Status = FALSE THEN
				temp_ver_value := FALSE;
			END_IF
		END_FOR
		
		IF GVL_HMI.HMI_SECTION_2_BEGIN_AUTOMATED_BUTTON.Live_Value AND temp_ver_value THEN
			GVL_HMI.ACTIVE_HMI_VIEW := 12;
		END_IF
		
	3:
	
		IF GVL_HMI.HMI_RESET_TEST_BUTTON.Live_Value THEN
			UNINITIALIZE();
		END_IF
		
		
	11:
		WRITE_IO_VALUES();
		Delay(IN := TRUE, PT := T#1S);
			
		IF Delay.Q THEN
			ExecuteSection1(StartTest := TRUE);
			
			IF ExecuteSection1.Done THEN
				LOG_SECTION1();
				GVL_HMI.ACTIVE_HMI_VIEW := 2;
			END_IF
		END_IF
		
	12: 
		WRITE_IO_VALUES();
		Delay1(IN := TRUE, PT := T#1S);
			
		IF Delay1.Q THEN
			ExecuteSection2(StartTest := TRUE);
				
			IF ExecuteSection2.Done THEN
				LOG_SECTION2();
				GVL_HMI.ACTIVE_HMI_VIEW := 3;
			END_IF
		END_IF

		
END_CASE

END_PROGRAM

// ---- POUs/FB_EXECUTE_SECTION1.TcPOU
FUNCTION_BLOCK FB_EXECUTE_SECTION1
VAR_INPUT
	StartTest : BOOL; // Tells this FB to start its checks
END_VAR

VAR_OUTPUT
	Done : BOOL; // Goes True when FB finishes its checks
END_VAR

VAR_IN_OUT
END_VAR

VAR
	i : INT;	
	state : INT; // internal step for the FB's state machine
	AddStep: INT;
END_VAR

IF StartTest THEN
	Done   := FALSE;
    CASE state OF
        0:
			// DIGITAL INPUTS
			FOR i := 0 TO CONSTANTS.SECTION1_NUM_DIG_TESTS - 1 DO
				IF GVL_IO_STRUCTS.IO_MAP_SECTION1_DIG[i].LIVE_BOOL = GVL_IO_STRUCTS.IO_MAP_SECTION1_DIG[i].EXPECTED_BOOL THEN
					GVL_IO_STRUCTS.IO_MAP_SECTION1_DIG[i].RESULT := 'PASS';
				ELSE
					GVL_IO_STRUCTS.IO_MAP_SECTION1_DIG[i].RESULT := 'FAIL';
				END_IF
			END_FOR
			
			FOR i := 0 TO CONSTANTS.SECTION1_NUM_HMI_TESTS -1 DO
				IF GVL_IO_STRUCTS.IO_MAP_SECTION1_HMI[i].LIVE_BOOL = GVL_IO_STRUCTS.IO_MAP_SECTION1_HMI[i].EXPECTED_BOOL THEN
					GVL_IO_STRUCTS.IO_MAP_SECTION1_HMI[i].RESULT := 'PASS';
				ELSE
					GVL_IO_STRUCTS.IO_MAP_SECTION1_HMI[i].RESULT := 'FAIL';
				END_IF
			END_FOR
			
			state := 999;
            
        999:
            // done
			Done := TRUE;
			state := 0;
        ;

    END_CASE;
ELSE
    // if StartTest = FALSE, reset
    Done   := FALSE;
    state  := 0;
END_IF

END_FUNCTION_BLOCK

// ---- POUs/FB_EXECUTE_SECTION2.TcPOU
FUNCTION_BLOCK FB_EXECUTE_SECTION2
VAR_INPUT
	StartTest : BOOL; // Tells this FB to start its checks
END_VAR

VAR_OUTPUT
	Done : BOOL; // Goes True when FB finishes its checks
END_VAR

VAR_IN_OUT
END_VAR

VAR
	i : INT;	
	state : INT; // internal step for the FB's state machine
	AddStep: INT;
END_VAR

IF StartTest THEN
	Done   := FALSE;
    CASE state OF
        0:
			// DIGITAL INPUTS
			FOR i := 0 TO CONSTANTS.SECTION2_NUM_DIG_TESTS - 1 DO
				IF GVL_IO_STRUCTS.IO_MAP_SECTION2_DIG[i].LIVE_BOOL = GVL_IO_STRUCTS.IO_MAP_SECTION2_DIG[i].EXPECTED_BOOL THEN
					GVL_IO_STRUCTS.IO_MAP_SECTION2_DIG[i].RESULT := 'PASS';
				ELSE
					GVL_IO_STRUCTS.IO_MAP_SECTION2_DIG[i].RESULT := 'FAIL';
				END_IF
			END_FOR
			
			FOR i := 0 TO CONSTANTS.SECTION2_NUM_HMI_TESTS -1 DO
				IF GVL_IO_STRUCTS.IO_MAP_SECTION2_HMI[i].LIVE_BOOL = GVL_IO_STRUCTS.IO_MAP_SECTION2_HMI[i].EXPECTED_BOOL THEN
					GVL_IO_STRUCTS.IO_MAP_SECTION2_HMI[i].RESULT := 'PASS';
				ELSE
					GVL_IO_STRUCTS.IO_MAP_SECTION2_HMI[i].RESULT := 'FAIL';
				END_IF
			END_FOR
			
			state := 999;
            
        999:
            // done
			Done := TRUE;
			state := 0;
        ;

    END_CASE;
ELSE
    // if StartTest = FALSE, reset
    Done   := FALSE;
    state  := 0;
END_IF

END_FUNCTION_BLOCK

// ---- POUs/UNINITIALIZE.TcPOU
FUNCTION UNINITIALIZE : BOOL
VAR_INPUT
END_VAR
VAR
	i : INT;
	in_progress : BOOL;
END_VAR


in_progress := TRUE;
	
FOR i := 0 TO CONSTANTS.SECTION1_NUM_DIG_TESTS - 1 DO
	GVL_IO_STRUCTS.IO_MAP_SECTION1_DIG[i].LIVE_BOOL := FALSE;
	GVL_IO_STRUCTS.IO_MAP_SECTION1_DIG[i].Result := 'FAIL';
END_FOR

FOR i := 0 TO CONSTANTS.SECTION1_NUM_HMI_TESTS - 1 DO
	GVL_IO_STRUCTS.IO_MAP_SECTION1_HMI[i].LIVE_BOOL := FALSE;
	GVL_IO_STRUCTS.IO_MAP_SECTION1_HMI[i].Result := 'FAIL';
END_FOR

FOR i := 0 TO CONSTANTS.SECTION2_NUM_DIG_TESTS - 1 DO
	GVL_IO_STRUCTS.IO_MAP_SECTION2_DIG[i].LIVE_BOOL := FALSE;
	GVL_IO_STRUCTS.IO_MAP_SECTION2_DIG[i].Result := 'FAIL';
END_FOR

FOR i := 0 TO CONSTANTS.SECTION2_NUM_HMI_TESTS - 1 DO
	GVL_IO_STRUCTS.IO_MAP_SECTION2_HMI[i].LIVE_BOOL := FALSE;
	GVL_IO_STRUCTS.IO_MAP_SECTION2_HMI[i].Result := 'FAIL';
END_FOR


FOR I := 0 TO GVL_LOGS.NUM_TESTS_LOGGED - 1 DO
	GVL_LOGS.TEST_RESULTS_ARRAY[i].Description := '';
	GVL_LOGS.TEST_RESULTS_ARRAY[i].Index := 0;
	GVL_LOGS.TEST_RESULTS_ARRAY[i].Result := '';
END_FOR

FOR i := 0 TO CONSTANTS.HMI_HOME_NUM_INSTRUCTIONS - 1 DO
		GVL_HMI.HMI_HOME_INSTRUCTIONS[i].Status := FALSE;
END_FOR

FOR i := 0 TO CONSTANTS.HMI_SECTION_1_NUM_INSTRUCTIONS - 1 DO
		GVL_HMI.HMI_SECTION_1_INSTRUCTIONS[i].Status := FALSE;
END_FOR

FOR i := 0 TO CONSTANTS.HMI_SECTION_2_NUM_INSTRUCTIONS - 1 DO
		GVL_HMI.HMI_SECTION_2_INSTRUCTIONS[i].Status := FALSE;
END_FOR

GVL_LOGS.NUM_TESTS_LOGGED := 0;

GVL_HMI.ACTIVE_HMI_VIEW := 0;


in_progress := FALSE;

Uninitialize := TRUE;

END_FUNCTION

// ---- POUs/INITIALIZE.TcPOU
FUNCTION INITIALIZE : BOOL
VAR_INPUT
END_VAR
VAR
	i : INT;
END_VAR


GVL_LOGS.NUM_TESTS_LOGGED := 0;


GVL_IO.SECTION1_DIG_INPUTS[0] := ADR(GVL_IO.J7_24V_Up);
GVL_IO.SECTION1_DIG_INPUTS[1] := ADR(GVL_IO.J7_24V_Us);
GVL_IO.SECTION1_DIG_INPUTS[2] := ADR(GVL_IO.J8_24V_Up);
GVL_IO.SECTION1_DIG_INPUTS[3] := ADR(GVL_IO.J8_24V_Us);
GVL_IO.SECTION1_DIG_INPUTS[4] := ADR(GVL_IO.J1_24V_Up);
GVL_IO.SECTION1_DIG_INPUTS[5] := ADR(GVL_IO.J1_24V_Us);
GVL_IO.SECTION1_DIG_INPUTS[6] := ADR(GVL_IO.J2_24V_Up);
GVL_IO.SECTION1_DIG_INPUTS[7] := ADR(GVL_IO.J2_24V_Us);
GVL_IO.SECTION1_DIG_INPUTS[8] := ADR(GVL_IO.J3_24V_Up);
GVL_IO.SECTION1_DIG_INPUTS[9] := ADR(GVL_IO.J3_24V_Us);
GVL_IO.SECTION1_DIG_INPUTS[10] := ADR(GVL_IO.J4_24V_Up);
GVL_IO.SECTION1_DIG_INPUTS[11] := ADR(GVL_IO.J4_24V_Us);
GVL_IO.SECTION1_DIG_INPUTS[12] := ADR(GVL_IO.J5_24V_Up);
GVL_IO.SECTION1_DIG_INPUTS[13] := ADR(GVL_IO.J5_24V_Us);
GVL_IO.SECTION1_DIG_INPUTS[14] := ADR(GVL_IO.J6_24V_Up);
GVL_IO.SECTION1_DIG_INPUTS[15] := ADR(GVL_IO.J6_24V_Us);
GVL_IO.SECTION1_DIG_INPUTS[16] := ADR(GVL_IO.SF1_MF_CONTINUITY);
GVL_IO.SECTION1_DIG_INPUTS[17] := ADR(GVL_IO.SF2_MF_CONTINUITY);
GVL_IO.SECTION1_DIG_INPUTS[18] := ADR(GVL_IO.SF4_Pull_Station);
GVL_IO.SECTION1_DIG_INPUTS[19] := ADR(GVL_IO.SF6_MGT_CONTINUITY);
GVL_IO.SECTION1_DIG_INPUTS[20] := ADR(GVL_IO.SF8_MGT_CONTINUITY);
GVL_IO.SECTION1_DIG_INPUTS[21] := ADR(GVL_IO.JB_Door_Switch);
GVL_IO.SECTION1_DIG_INPUTS[22] := ADR(GVL_IO.JB_DCDCS_OK);
GVL_IO.SECTION1_DIG_INPUTS[23] := ADR(GVL_IO.JB_PSU2_OK);


GVL_IO.SECTION2_DIG_INPUTS[0] := ADR(GVL_IO.SF4_Pull_Station);
GVL_IO.SECTION2_DIG_INPUTS[1] := ADR(GVL_IO.JB_Door_Switch);
GVL_IO.SECTION2_DIG_INPUTS[2] := ADR(GVL_IO.JB_PSU1_OK);
GVL_IO.SECTION2_DIG_INPUTS[3] := ADR(GVL_IO.J7_24V_Up);
GVL_IO.SECTION2_DIG_INPUTS[4] := ADR(GVL_IO.J7_24V_Us);
GVL_IO.SECTION2_DIG_INPUTS[5] := ADR(GVL_IO.J8_24V_Up);
GVL_IO.SECTION2_DIG_INPUTS[6] := ADR(GVL_IO.J8_24V_Us);
GVL_IO.SECTION2_DIG_INPUTS[7] := ADR(GVL_IO.J1_24V_Up);
GVL_IO.SECTION2_DIG_INPUTS[8] := ADR(GVL_IO.J1_24V_Us);
GVL_IO.SECTION2_DIG_INPUTS[9] := ADR(GVL_IO.J2_24V_Up);
GVL_IO.SECTION2_DIG_INPUTS[10] := ADR(GVL_IO.J2_24V_Us);
GVL_IO.SECTION2_DIG_INPUTS[11] := ADR(GVL_IO.J3_24V_Up);
GVL_IO.SECTION2_DIG_INPUTS[12] := ADR(GVL_IO.J3_24V_Us);
GVL_IO.SECTION2_DIG_INPUTS[13] := ADR(GVL_IO.J4_24V_Up);
GVL_IO.SECTION2_DIG_INPUTS[14] := ADR(GVL_IO.J4_24V_Us);
GVL_IO.SECTION2_DIG_INPUTS[15] := ADR(GVL_IO.J5_24V_Up);
GVL_IO.SECTION2_DIG_INPUTS[16] := ADR(GVL_IO.J5_24V_Us);
GVL_IO.SECTION2_DIG_INPUTS[17] := ADR(GVL_IO.J6_24V_Up);
GVL_IO.SECTION2_DIG_INPUTS[18] := ADR(GVL_IO.J6_24V_Us);


INITIALIZE := TRUE;

END_FUNCTION

// ---- POUs/WRITE_IO_VALUES.TcPOU
FUNCTION WRITE_IO_VALUES : BOOL
VAR_INPUT
END_VAR
VAR
	i : INT;
END_VAR


// Write Values to IO Structures


// WRITE VALUES TO SECTION 1 Digital Input VARIABLES
FOR i := 0 TO CONSTANTS.SECTION1_NUM_DIG_TESTS - 1 DO
	GVL_IO_STRUCTS.IO_MAP_SECTION1_DIG[i].LIVE_BOOL := GVL_IO.SECTION1_DIG_INPUTS[i]^;
END_FOR

// WRITE VALUES TO Section 1 HMI INPUT TESTS

GVL_IO_STRUCTS.IO_MAP_SECTION1_HMI[0].LIVE_BOOL := GVL_HMI.HMI_SECTION_1_INSTRUCTIONS[0].Status;
GVL_IO_STRUCTS.IO_MAP_SECTION1_HMI[1].LIVE_BOOL := GVL_HMI.HMI_SECTION_1_INSTRUCTIONS[1].Status;
GVL_IO_STRUCTS.IO_MAP_SECTION1_HMI[2].LIVE_BOOL := GVL_HMI.HMI_SECTION_1_INSTRUCTIONS[2].Status;
GVL_IO_STRUCTS.IO_MAP_SECTION1_HMI[3].LIVE_BOOL := GVL_HMI.HMI_SECTION_1_INSTRUCTIONS[3].Status;


// WRITE VALUES TO SECTION 2 Digital Input Variables
FOR i := 0 TO CONSTANTS.SECTION2_NUM_DIG_TESTS - 1 DO
	GVL_IO_STRUCTS.IO_MAP_SECTION2_DIG[i].LIVE_BOOL := GVL_IO.SECTION2_DIG_INPUTS[i]^;
END_FOR


GVL_IO_STRUCTS.IO_MAP_SECTION2_HMI[0].LIVE_BOOL := GVL_HMI.HMI_SECTION_2_INSTRUCTIONS[4].Status;
GVL_IO_STRUCTS.IO_MAP_SECTION2_HMI[1].LIVE_BOOL := GVL_HMI.HMI_SECTION_2_INSTRUCTIONS[5].Status;
GVL_IO_STRUCTS.IO_MAP_SECTION2_HMI[2].LIVE_BOOL := GVL_HMI.HMI_SECTION_2_INSTRUCTIONS[6].Status;




// Write Values to other test variables


(*
GVL_IO_STRUCTS.FIRE_ALRM_P5.LIVE_BOOL := GVL_IO.C2_P2;
GVL_IO_STRUCTS.JB_CARD_Us.LIVE_BOOL := GVL_IO.JB_1914_Us;
GVL_IO_STRUCTS.JB_CARD_Up.LIVE_BOOL := GVL_IO.JB_1914_Up;
GVL_IO_STRUCTS.FIRE_PULL_P4.LIVE_BOOL := GVL_IO.C3_P1;
GVL_IO_STRUCTS.Us_24V_5.LIVE_BOOL := GVL_IO.C3_P2;
GVL_IO_STRUCTS.Up_24V_5.LIVE_BOOL := GVL_IO.C3_P3;
GVL_IO_STRUCTS.Us_24V_1.LIVE_BOOL := GVL_IO.C3_P4;
GVL_IO_STRUCTS.Up_24V_1.LIVE_BOOL := GVL_IO.C3_P5;
GVL_IO_STRUCTS.Us_24V_2.LIVE_BOOL := GVL_IO.C3_P6;
GVL_IO_STRUCTS.Up_24V_2.LIVE_BOOL := GVL_IO.C3_P7;
GVL_IO_STRUCTS.Us_24V_3.LIVE_BOOL := GVL_IO.C4_P1;
GVL_IO_STRUCTS.Up_24V_3.LIVE_BOOL := GVL_IO.C4_P2;
GVL_IO_STRUCTS.Us_24V_4.LIVE_BOOL := GVL_IO.C4_P3;
GVL_IO_STRUCTS.Up_24V_4.LIVE_BOOL := GVL_IO.C4_P4;
GVL_IO_STRUCTS.Us_24V_6.LIVE_BOOL := GVL_IO.C4_P5;
GVL_IO_STRUCTS.Up_24V_6.LIVE_BOOL := GVL_IO.C4_P6;
GVL_IO_STRUCTS.PHONE_P2.LIVE_BOOL := GVL_IO.C4_P7;
GVL_IO_STRUCTS.PHONE_P1.LIVE_BOOL := GVL_IO.C4_P8;
GVL_IO_STRUCTS.MGT_P6.LIVE_BOOL := GVL_IO.C5_P1;
GVL_IO_STRUCTS.MGT_P8.LIVE_BOOL := GVL_IO.C5_P2;
GVL_IO_STRUCTS.LIGHT_24V_Us_1.LIVE_BOOL := GVL_IO.C5_P3;
GVL_IO_STRUCTS.LIGHT_24V_Up_1.LIVE_BOOL := GVL_IO.C5_P4;
GVL_IO_STRUCTS.LIGHT_24V_Us_2.LIVE_BOOL := GVL_IO.C5_P5;
GVL_IO_STRUCTS.LIGHT_24V_Up_2.LIVE_BOOL := GVL_IO.C5_P6;
*)

END_FUNCTION

// ---- POUs/LOG_SECTION1.TcPOU
FUNCTION LOG_SECTION1 : BOOL
VAR_INPUT
END_VAR
VAR
	i : INT;
	j : INT;
	dig_start_index : INT;
	dig_end_index : INT;
	
	hmi_start_index : INT;
	hmi_end_index : INT;
	
	Done : BOOL;
END_VAR

Done := FALSE;

dig_start_index := GVL_LOGS.NUM_TESTS_LOGGED;
dig_end_index := dig_start_index + CONSTANTS.SECTION1_NUM_DIG_TESTS-1;

// SECTION 1 DIGITAL INPUTS
FOR i := dig_start_index TO dig_end_index DO
	j := i - dig_start_index;
	GVL_LOGS.TEST_RESULTS_ARRAY[i].DESCRIPTION := GVL_IO_STRUCTS.IO_MAP_SECTION1_DIG[j].DESCRIPTION;
	GVL_LOGS.TEST_RESULTS_ARRAY[i].INDEX := i;
	GVL_LOGS.TEST_RESULTS_ARRAY[i].RESULT := GVL_IO_STRUCTS.IO_MAP_SECTION1_DIG[j].RESULT;
	GVL_LOGS.NUM_TESTS_LOGGED := GVL_LOGS.NUM_TESTS_LOGGED + 1;
END_FOR

hmi_start_index := GVL_LOGS.NUM_TESTS_LOGGED;
hmi_end_index := hmi_start_index + CONSTANTS.SECTION1_NUM_HMI_TESTS-1;

FOR i := hmi_start_index TO hmi_end_index DO
	j := i - hmi_start_index;
	GVL_LOGS.TEST_RESULTS_ARRAY[i].DESCRIPTION := GVL_IO_STRUCTS.IO_MAP_SECTION1_HMI[j].DESCRIPTION;
	GVL_LOGS.TEST_RESULTS_ARRAY[i].INDEX := i;
	GVL_LOGS.TEST_RESULTS_ARRAY[i].RESULT := GVL_IO_STRUCTS.IO_MAP_SECTION1_HMI[j].RESULT;
	GVL_LOGS.NUM_TESTS_LOGGED := GVL_LOGS.NUM_TESTS_LOGGED + 1;
END_FOR

Done := TRUE;

END_FUNCTION

// ---- POUs/LOG_SECTION2.TcPOU
FUNCTION LOG_SECTION2 : BOOL
VAR_INPUT
END_VAR
VAR
	i : INT;
	j : INT;
	start_index : INT;
	end_index : INT;
	
	hmi_start_index : INT;
	hmi_end_index : INT;
END_VAR
VAR_OUTPUT
	Done : BOOL;
END_VAR

Done := FALSE;

start_index := GVL_LOGS.NUM_TESTS_LOGGED;
end_index := start_index + CONSTANTS.SECTION2_NUM_DIG_TESTS-1;

// SECTION 2 DIGITAL INPUTS
FOR i := start_index TO end_index DO
	j := i - start_index;
	GVL_LOGS.TEST_RESULTS_ARRAY[i].DESCRIPTION := GVL_IO_STRUCTS.IO_MAP_SECTION2_DIG[j].DESCRIPTION;
	GVL_LOGS.TEST_RESULTS_ARRAY[i].INDEX := i;
	GVL_LOGS.TEST_RESULTS_ARRAY[i].RESULT := GVL_IO_STRUCTS.IO_MAP_SECTION2_DIG[j].RESULT;
	GVL_LOGS.NUM_TESTS_LOGGED := GVL_LOGS.NUM_TESTS_LOGGED + 1;
END_FOR

hmi_start_index := GVL_LOGS.NUM_TESTS_LOGGED;
hmi_end_index := hmi_start_index + CONSTANTS.SECTION2_NUM_HMI_TESTS-1;

FOR i := hmi_start_index TO hmi_end_index DO
	j := i - hmi_start_index;
	GVL_LOGS.TEST_RESULTS_ARRAY[i].DESCRIPTION := GVL_IO_STRUCTS.IO_MAP_SECTION2_HMI[j].DESCRIPTION;
	GVL_LOGS.TEST_RESULTS_ARRAY[i].INDEX := i;
	GVL_LOGS.TEST_RESULTS_ARRAY[i].RESULT := GVL_IO_STRUCTS.IO_MAP_SECTION2_HMI[j].RESULT;
	GVL_LOGS.NUM_TESTS_LOGGED := GVL_LOGS.NUM_TESTS_LOGGED + 1;
END_FOR

Done := TRUE;

END_FUNCTION
